FUNCTION_BLOCK FB_HeatPumpSystem_HNHT EXTENDS FB_SystemContinous
VAR_INPUT
END_VAR
VAR_OUTPUT
END_VAR
VAR
	//Vitocal 350-G heat pump
	HeatPump : FB_HeatPump;
	
	//valves
	ST_RV342DefaultParameters : ST_MixingValveDefaultParameters := (fControllerAmplification := 5, tControllerIntegralTime := T#100S, tTaskCycleTime := GlobalVariables.tTaskCycleTime_MAIN, tCtrlCycleTime := GlobalVariables.tCtrlCycleTime_MAIN, fOffsetTerminal := 2900);;
	ST_RV242DefaultParameters : ST_MixingValveDefaultParameters := (fControllerAmplification := 10, tControllerIntegralTime := T#100S, tTaskCycleTime := GlobalVariables.tTaskCycleTime_MAIN, tCtrlCycleTime := GlobalVariables.tCtrlCycleTime_MAIN, fOffsetTerminal := 3500);
	ST_SV_HNLT_DefaultParameters : ST_DiscreteValveDefaultParameters := (nFeedback := 0);		
	RV342 : FB_MixingValve := (ST_DefaultParameters := ST_RV342DefaultParameters);
	RV242 : FB_MixingValve := (ST_DefaultParameters := ST_RV242DefaultParameters);	
	SV_HNLT : FB_DiscreteValve := (ST_DefaultParameters := ST_SV_HNLT_DefaultParameters);	
	
	//pump
	stPU242DefaultParameters : ST_PumpGrundfosMagna3DefaultParameters := (tTaskCycleTime := GlobalVariables.tTaskCycleTime_MAIN, tCtrlCycleTime := GlobalVariables.tCtrlCycleTime_MAIN, bExternalTemperatureSensor := TRUE);
	PU242 : FB_PumpGrundfosMagna3 := (ST_DefaultParameters := stPU242DefaultParameters);
	
	//internal variables
	bSetStatusOn_HeatPump : BOOL;
	bSetStatusOn_PU242 : BOOL;
	bSetStatusOn_RV342 : BOOL;
	bSetStatusOn_RV242 : BOOL;
	bSetStatusOn_SV_HNLT : BOOL;
	fTemperatureSetPoint_RV242 : REAL;
	
	// timer for SV441, SV442
	bStartTimer_SV : BOOL;
	Timer_SV : TON;
	
	// timer for heat pump
	bStartTimer_HeatPump : BOOL;
	Timer_HeatPump : TON;
	
	//error variable for temperature TS242
	Controller_TS242_Error : FB_CTRL_2POINT;
	Controller_TS242_Error_Parameters : ST_CTRL_2POINT_PARAMS;

	//sensors
	TS242 : FB_TemperatureSensor; //inlet temperature evaporator
	WMZ342 : FB_MollineEHeatCounter;
END_VAR

MAIN();
//use timer for cool down during ramp up
Timer_SV(IN := bStartTimer_SV,
	PT := T#30S);
Timer_HeatPump(IN := bStartTimer_HeatPump,
	PT := T#180S);

//valves
SV_HNLT.GetState_BI();
SV_HNLT(bSetStatusOnAutomatic := bSetStatusOn_SV_HNLT,
		bAlgorithmPermission := bAlgorithmPermission);
SV_HNLT.SetState_BO();

//heat pump
HeatPump.GetState();
HeatPump(bSetStatusOnAutomatic := bSetStatusOn_HeatPump,
	bAlgorithmPermission := bAlgorithmPermission,
	fSetPointAutomatic := fSetPoint);
HeatPump.SetState();

//pump
PU242.GetState_Profibus();
PU242(bSetStatusOnAutomatic := bSetStatusOn_PU242,
	fSetPointAutomatic := 100,
	bAlgorithmPermission := bAlgorithmPermission,
	nControlModeAutomatic := 0);
PU242.SetState_Profibus();

//valves
RV242.GetState_AI();
RV242(bSetStatusOnAutomatic := bSetStatusOn_RV242,
	bAlgorithmPermission := bAlgorithmPermission,
	fSetPointAutomatic := fTemperatureSetPoint_RV242,
	fTemperatureExternal := TS242.fTemperature,
	nControlModeAutomatic := 1);
RV242.SetState_AO();

RV342.GetState_AI();
RV342(bSetStatusOnAutomatic := bSetStatusOn_RV342,
	bAlgorithmPermission := bAlgorithmPermission,
	fSetPointAutomatic := 100,
	nControlModeAutomatic := 0);
RV342.SetState_AO();

//sensors
WMZ342(aHeatCounterTelegramm := aTelegramm_WMZ342);
TS242();
TS242.GetState_AI();

METHOD PROTECTED  CheckError : BOOL
VAR_INPUT
END_VAR
VAR_OUTPUT
	bError : BOOL;
END_VAR
Controller_TS242_Error_Parameters.fHysteresisRange := 2;
Controller_TS242_Error_Parameters.tCtrlCycleTime := GlobalVariables.tCtrlCycleTime_MAIN;
Controller_TS242_Error_Parameters.tTaskCycleTime := GlobalVariables.tTaskCycleTime_MAIN;

Controller_TS242_Error(fSetpointValue := 10,
	fActualValue := TS242.fTemperature,
	eMode := eCTRL_MODE_ACTIVE,
	stParams := Controller_TS242_Error_Parameters);

bError := HeatPump.bError OR PU242.bError OR Controller_TS242_Error.bOut;
END_METHOD

METHOD PROTECTED  Operational : BOOL
VAR_INPUT
END_VAR
VAR_OUTPUT
	bSwitchToWorking : BOOL := FALSE;
END_VAR
bSetStatusOn_PU242 := TRUE;

IF PU242.bStatusOn THEN
	bStartTimer_SV := TRUE;
	fTemperatureSetPoint_RV242 := 100;// open RV242 for cooling
	IF Timer_SV.Q THEN
		bStartTimer_SV := FALSE; //resets timer	
		bSetStatusOn_HeatPump := TRUE;
		bStartTimer_HeatPump := TRUE;
		IF Timer_HeatPump.Q THEN		
			bStartTimer_HeatPump := FALSE;
			bSwitchToWorking := TRUE;
		END_IF
	END_IF;
END_IF;
END_METHOD

METHOD PROTECTED  RampDown : BOOL
VAR_INPUT
END_VAR
VAR_OUTPUT
	bRampDownFinished : BOOL := FALSE;
END_VAR
bSetStatusOn_HeatPump := FALSE;

IF NOT HeatPump.bStatusOn  THEN
	bSetStatusOn_PU242 := FALSE;
	IF NOT PU242.bStatusOn  THEN
		bSetStatusOn_RV242 := FALSE;
		bSetStatusOn_RV342 := FALSE;
		bSetStatusOn_SV_HNLT := FALSE;
	
		IF RV242.fOperatingPoint<10 AND RV342.fOperatingPoint<10 THEN
			bRampDownFinished := TRUE;
		END_IF
	END_IF;
END_IF
END_METHOD

METHOD PROTECTED  RampUp : BOOL
VAR_INPUT
END_VAR
VAR_OUTPUT
	bRampUpFinished : BOOL := FALSE;
END_VAR
bSetStatusOn_RV242 := TRUE;
bSetStatusOn_RV342 := TRUE;
fTemperatureSetPoint_RV242 := 100;
bSetStatusOn_SV_HNLT := FALSE; //connects CN to heat pump
IF RV342.fOperatingPoint>80 THEN
	bRampUpFinished := TRUE;
END_IF
END_METHOD

METHOD PROTECTED   SetSetPointLimits : BOOL
VAR_INPUT
END_VAR
//heat pump has no continous setpoint (limits are not used) but must be implemented because of abstract method
aSetPointLimits[1] := 10;
aSetPointLimits[2] := 100;
END_METHOD

METHOD PROTECTED  SetState : BOOL
VAR_INPUT
END_VAR
VAR_OUTPUT
END_VAR
fOperatingPoint := WMZ342.fFeedTemperature;

controlState.bStatusOn := HeatPump.bStatusOn;
setPointState.aSetPointLimits := aSetPointLimits;
setPointState.fSetPoint := fSetPoint;
setPointState.fOperatingPoint := fOperatingPoint;
setPointState.sSetPointUnit := 'degreeC';
setPointState.sOperatingPointUnit := 'degreeC';
END_METHOD

METHOD PROTECTED  Working : BOOL
VAR_INPUT
END_VAR
VAR_OUTPUT
	bSwitchToOperational : BOOL := FALSE;
END_VAR
bSetStatusOn_SV_HNLT := TRUE; //connects HNLT to heat pump
fTemperatureSetPoint_RV242 := 20;// temperature setpoint for heating
END_METHOD

END_FUNCTION_BLOCK

(* stored: Version 1.1.0.1, ProductVersion 3.1.4024.10
   POU FB_HeatPumpSystem_HNHT: Id {6a406844-89d7-4db6-814d-0ca6a50f7081}, SpecialFunc None
   Method CheckError: Id {c81c127c-2dfa-453f-9842-92a23e6502aa}
   Method Operational: Id {23ee8fd7-999e-4774-94e8-1d99d6bd9b1b}
   Method RampDown: Id {3d77f4ba-35c2-425d-b53f-83f5a3e83c2b}
   Method RampUp: Id {d6507405-d735-45e3-a15b-80e07b56ab86}
   Method SetSetPointLimits: Id {afedc7e1-d1ba-48f7-b310-e0f65f399073}
   Method SetState: Id {12063f21-1e93-47c1-bde8-a30ea5d90a5b}
   Method Working: Id {87f552f2-0115-4afb-a2e6-1e42102018d3} *)
